FUNCTION_BLOCK AX_CLIENT_1_0 (* Send a BOOL from an AX adapter as a remote OPC-UA write via CLIENT_1_0, buffered with a E_D_FF *)
  (* Standard: 61499-2; Description: Copyright (c) 2026 HR Agrartechnik GmbH This program and the accompanying materials are made available under the terms of the Eclipse Public License 2.0 which is available at https://www.eclipse.org/legal/epl-2.0/ SPDX-License-Identifier: EPL-2.0 *)
  (* Version 1.0, 2026-08-27, Franz Höpfinger, HR Agrartechnik GmbH, initial API and implementation and/or initial documentation *)
  PACKAGE adapter::net;
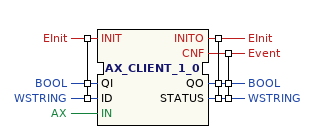
  EVENT_INPUT
    INIT : EInit WITH QI, ID; (* Initialization *)
  END_EVENT
  EVENT_OUTPUT
    INITO : EInit WITH QO, STATUS; (* Initialization Confirm *)
    CNF WITH QO, STATUS; (* Data was sent *)
  END_EVENT
  VAR_INPUT
    QI : BOOL;
    ID : WSTRING;
  END_VAR
  VAR_OUTPUT
    QO : BOOL;
    STATUS : WSTRING;
  END_VAR
  SOCKETS
    IN : adapter::types::unidirectional::AX; (* BOOL to send *)
  END_SOCKETS
  FBS
    E_D_FF : iec61499::events::E_D_FF;
    CLIENT_1_0 : iec61499::net::CLIENT_1_0;
  END_FBS
  EVENT_CONNECTIONS
    CLIENT_1_0.INITO TO INITO;
    CLIENT_1_0.CNF TO CNF;
    IN.E1 TO E_D_FF.CLK;
    E_D_FF.EO TO CLIENT_1_0.REQ;
    INIT TO CLIENT_1_0.INIT;
  END_CONNECTIONS
  DATA_CONNECTIONS
    CLIENT_1_0.QO TO QO;
    CLIENT_1_0.STATUS TO STATUS;
    IN.D1 TO E_D_FF.D;
    E_D_FF.Q TO CLIENT_1_0.SD_1;
    QI TO CLIENT_1_0.QI;
    ID TO CLIENT_1_0.ID;
  END_CONNECTIONS
END_FUNCTION_BLOCK
